FUNCTION_BLOCK FB_Skill_Load
VAR_INPUT
END_VAR
VAR_OUTPUT
END_VAR
VAR
END_VAR

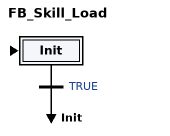
INITIAL_STEP Init:
END_STEP
TRANSITION FROM Init TO Init
    := TRUE;
END_TRANSITION

END_FUNCTION_BLOCK

(* stored: Version 1.1.0.1, ProductVersion 3.1.4026.18
   POU FB_Skill_Load: Id {11b4d487-9b5c-4e3b-b43a-7da8db436746}, SpecialFunc None *)
